FUNCTION_BLOCK RgbController
VAR
	_Red		AT %Q*	: BOOL;
	_Green		AT %Q*	: BOOL;
	_Blue		AT %Q*	: BOOL;
END_VAR

METHOD SetCustom : BOOL
VAR_INPUT
	Red		: BOOL;
	Green	: BOOL;
	Blue	: BOOL;
END_VAR
_Red := Red;
_Green := Green;
_Blue := Blue;
END_METHOD

METHOD SetWhite : BOOL
VAR_INPUT
END_VAR
_Red := TRUE;
_Green := TRUE;
_Blue := TRUE;
END_METHOD

METHOD TurnOff : BOOL
VAR_INPUT
END_VAR
_Red := FALSE;
_Green := FALSE;
_Blue := FALSE;
END_METHOD

END_FUNCTION_BLOCK

(* stored: Version 1.1.0.1
   POU RgbController: Id {8c2ea173-7e7f-4e6f-890a-03ebba81d070}, SpecialFunc None
   Method SetCustom: Id {efd4df41-d278-49f1-839f-91a8eacd7959}
   Method SetWhite: Id {cc5e42d6-471d-4be2-858f-e2fbc049f843}
   Method TurnOff: Id {c8d11621-676e-4fec-a7b3-24bba1f2df69} *)
